FUNCTION "FC_Val_Max_Calc" : Void
{ S7_Optimized_Access := 'TRUE' }
VERSION : 0.1
   VAR_INPUT
      Grandeur : Real;
      Grandeur_Max : Real;
   END_VAR

   VAR_OUTPUT
      Val_Max_Cal : Real;
   END_VAR


BEGIN
	#Val_Max_Cal := (#Grandeur / #Grandeur_Max) * 100;
END_FUNCTION

